// SIMATIC S7-200 project (STEP 7-Micro/WIN), CPU 221 REL 01.10

ORGANIZATION_BLOCK MAIN:OB1
TITLE=PROGRAM COMMENTS  标准报警电路
BEGIN
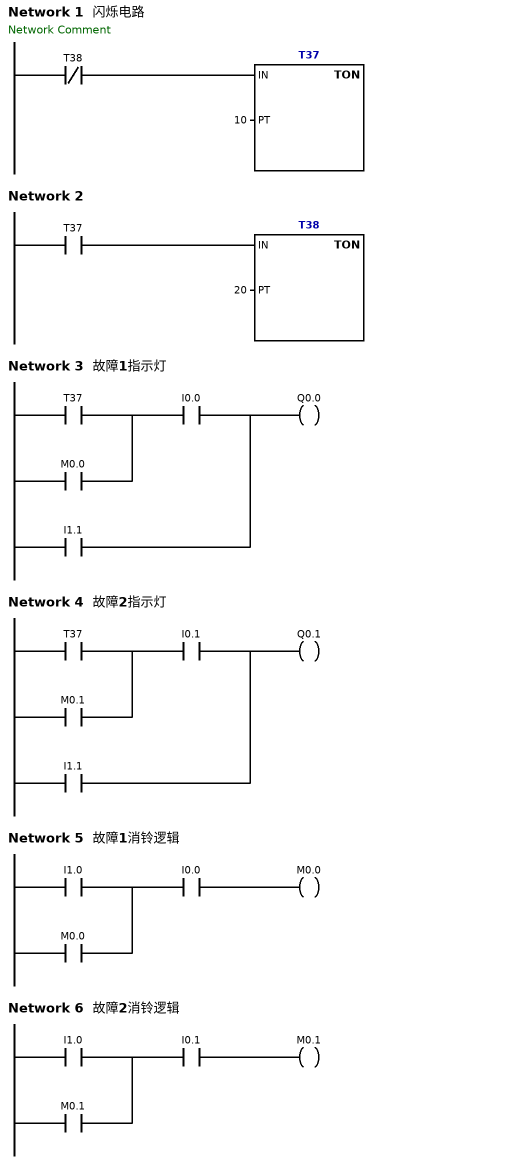
Network 1 // 闪烁电路
// Network Comment
LDN    T38
TON    T37, 10
Network 2
LD     T37
TON    T38, 20
Network 3 // 故障1指示灯
LD     T37
O      M0.0
A      I0.0
O      I1.1
=      Q0.0
Network 4 // 故障2指示灯
LD     T37
O      M0.1
A      I0.1
O      I1.1
=      Q0.1
Network 5 // 故障1消铃逻辑
LD     I1.0
O      M0.0
A      I0.0
=      M0.0
Network 6 // 故障2消铃逻辑
LD     I1.0
O      M0.1
A      I0.1
=      M0.1
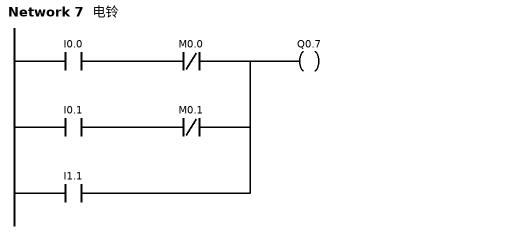
Network 7 // 电铃
LD     I0.0
AN     M0.0
LD     I0.1
AN     M0.1
OLD
O      I1.1
=      Q0.7
END_ORGANIZATION_BLOCK
